// Mitsubishi GX Works2 project: k03   PLC: Q02/Q02H

PROGRAM MAIN
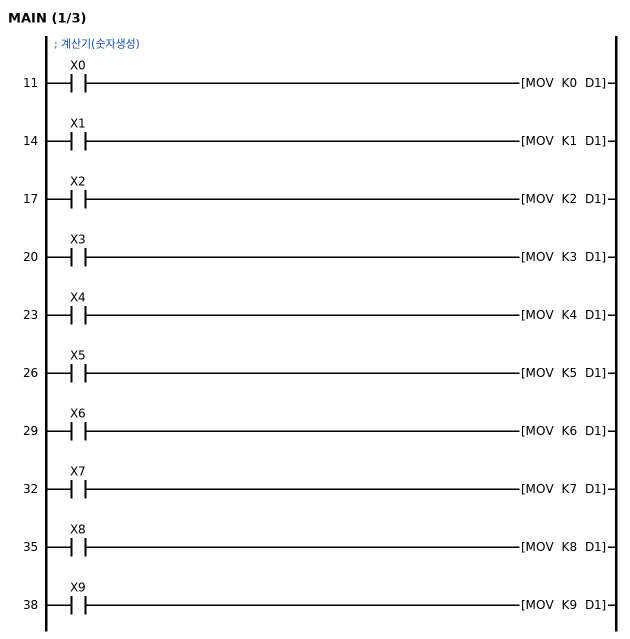
; 계산기(숫자생성)
11    LD      X0
      MOV     K0 D1
14    LD      X1
      MOV     K1 D1
17    LD      X2
      MOV     K2 D1
20    LD      X3
      MOV     K3 D1
23    LD      X4
      MOV     K4 D1
26    LD      X5
      MOV     K5 D1
29    LD      X6
      MOV     K6 D1
32    LD      X7
      MOV     K7 D1
35    LD      X8
      MOV     K8 D1
38    LD      X9
      MOV     K9 D1
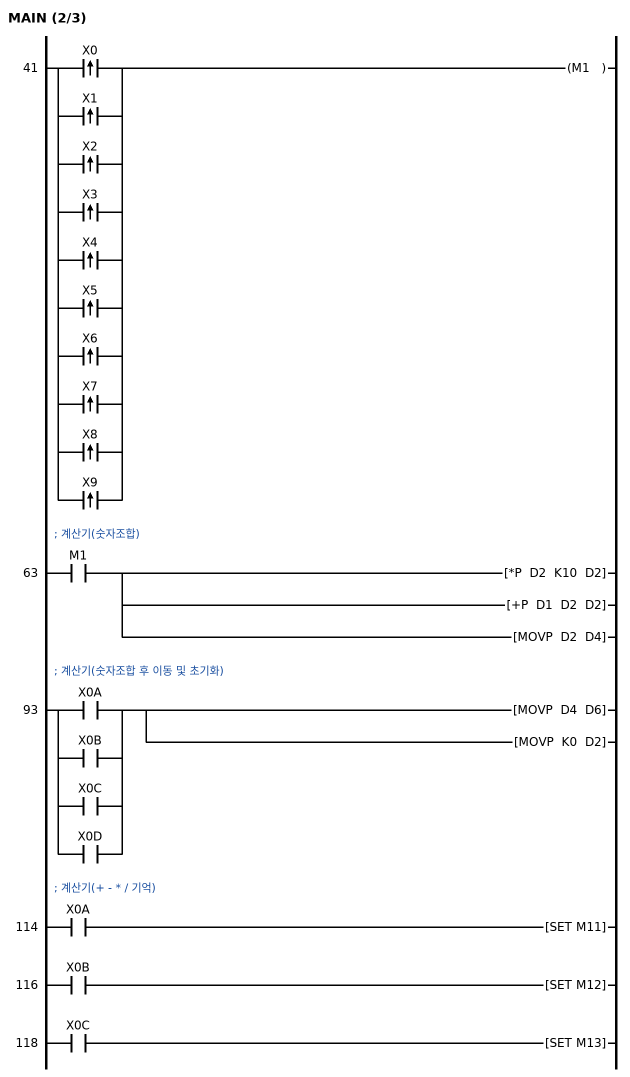
41    LDP     X0
      ORP     X1
      ORP     X2
      ORP     X3
      ORP     X4
      ORP     X5
      ORP     X6
      ORP     X7
      ORP     X8
      ORP     X9
      OUT     M1
; 계산기(숫자조합)
63    LD      M1
      *P      D2 K10 D2
      +P      D1 D2 D2
      MOVP    D2 D4
; 계산기(숫자조합 후 이동 및 초기화)
93    LD      X0A
      OR      X0B
      OR      X0C
      OR      X0D
      MOVP    D4 D6
      MOVP    K0 D2
; 계산기(+ - * / 기억)
114   LD      X0A
      SET     M11
116   LD      X0B
      SET     M12
118   LD      X0C
      SET     M13
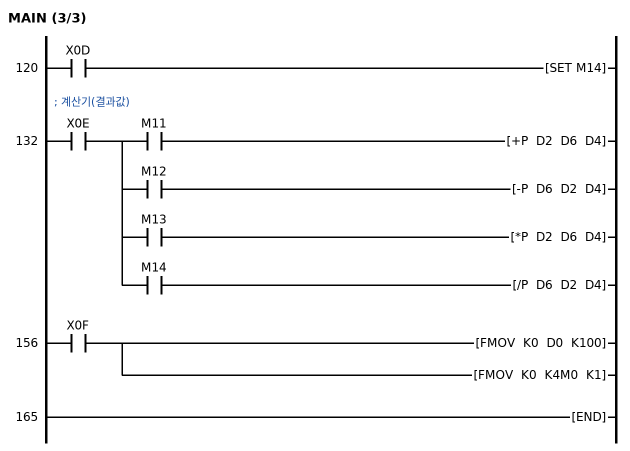
120   LD      X0D
      SET     M14
; 계산기(결과값)
132   LD      X0E
      MPS
      AND     M11
      +P      D2 D6 D4
      MRD
      AND     M12
      -P      D6 D2 D4
      MRD
      AND     M13
      *P      D2 D6 D4
      MPP
      AND     M14
      /P      D6 D2 D4
156   LD      X0F
      FMOV    K0 D0 K100
      FMOV    K0 K4M0 K1
165   END
END_PROGRAM
